FUNCTION_BLOCK EM_DockingInterface EXTENDS EM_Base IMPLEMENTS I_EM_DockingInterface
VAR_INPUT
//Inputs
	i_ref_stSettings : REFERENCE TO ST_SettingsDockingInterface;
	
	//--i_bIlckDockingClampsToClose : BOOL := TRUE; //TRUE = Interlocked
	//--i_bIlckDockingClampsToOpen : BOOL := TRUE; //TRUE = Interlocked
	//--i_bIlckUnlockingPinsToLock : BOOL := TRUE; //TRUE = Interlocked
	//--i_bIlckUnlockingPinsToRelease : BOOL := TRUE; //TRUE = Interlocked
	
	// External interlocks (from outside this EM)
	i_fbExtIlckDockingClampsToClose : FB_Interlock;
	i_fbExtIlckDockingClampsToOpen : FB_Interlock;
	i_fbExtIlckUnlockingPinsToLock : FB_Interlock;
	i_fbExtIlckUnlockingPinsToRelease : FB_Interlock;
	
	i_fbExtIlckInnerDoorOpen : FB_Interlock;
	i_fbExtIlckInnerDoorClose : FB_Interlock;
	
	
	
	i_refTB : REFERENCE TO OBJ_Carrier;	//Mogelijk voor uiteindelijke machine, voor de FUMO's is dit nog niet echt relevant
	//??i_refITF_TB : REFERENCE TO I_Carrier;
END_VAR

VAR_OUTPUT
	q_bStaWarning : BOOL;
END_VAR

VAR
//------------------------------------------//
//Control Modules (Devices)
	s_cmDockingClampsUpper : CM_ValveWithDoubleFB; // Off = Open, On = Close
	s_cmDockingClampsLower : CM_ValveWithDoubleFB; // Off = Open, On = Close
	
	s_cmUnlockingPinUpper : CM_ValveWithFB; // Off = Lock, On = Release
	s_cmUnlockingPinLower : CM_ValveWithFB; // Off = Lock, On = Release
	
	s_cmDoorOpener : CM_ValveWithFB; // Off = Close, On = Open
	s_cmDoorShutter : CM_ValveWithFB; // Off = Open, On = Close
	
//Interlocks	
fbIlckHandlerDockingClampsOpen : FB_InterlockHandler;
fbIlckHandlerDockingClampsClose : FB_InterlockHandler;
fbIlckHandlerUnlockingPinsLock : FB_InterlockHandler;
fbIlckHandlerUnlockingPinsRelease : FB_InterlockHandler;
fbIlckHandlerDoorOpenerClose : FB_InterlockHandler;
fbIlckHandlerDoorOpenerOpen : FB_InterlockHandler;
fbIlckHandlerDoorShutterClose : FB_InterlockHandler;
fbIlckHandlerDoorShutterOpen : FB_InterlockHandler;

//--fbInterlockHandlerDockTB : FB_InterlockHandler;
//--fbInterlockHandlerUndockTB : FB_InterlockHandler;
//--fbInterlockHandlerOpenInnerDoor : FB_InterlockHandler;
//--fbInterlockHandlerCloseInnerDoor : FB_InterlockHandler;	


	
//------------------------------------------//

//------------------------------------------//
//Inputs
	s_diStaDoorAlmostClosed : FB_DigInput;
		
//------------------------------------------//
	
//------------------------------------------//
//Outputs
	s_doCmdClampsUpperHighPressure : FB_DigOutput_2;
	s_doCmdClampsLowerHighPressure : FB_DigOutput_2;

//------------------------------------------//

//Requests
	s_bReqDockBox : BOOL := FALSE;
	s_bReqUndockBox : BOOL := FALSE;
	s_bReqOpenInnerDoor : BOOL := FALSE;
	s_bReqCloseInnerDoor : BOOL := FALSE;
	s_bReqDockingClampsUpperHighPressure : BOOL := FALSE; // True = high pressure
	s_bReqDockingClampsLowerHighPressure : BOOL := FALSE; // True = high pressure
	
	s_bOverruleInterlocks : BOOL := FALSE;
	
//Properties
	s_bStaDocked : BOOL := FALSE;
	s_bStaUndocked : BOOL := FALSE;
	
	s_bStaDockingClampsClosed : BOOL := FALSE;
	s_bStaDockingClampsOpened : BOOL := FALSE;
	s_bStaDockingClampsUpperClosed : BOOL := FALSE;
	s_bStaDockingClampsUpperOpened : BOOL := FALSE;
	s_bStaDockingClampsLowerClosed : BOOL := FALSE;
	s_bStaDockingClampsLowerOpened : BOOL := FALSE;
	
	s_bStaLockingPinUpperReleased : BOOL := FALSE;
	s_bStaLockingPinUpperLocked : BOOL := FALSE;
	s_bStaLockingPinLowerReleased : BOOL := FALSE;
	s_bStaLockingPinLowerLocked : BOOL := FALSE;
		
	s_bStaDoorOpenerOpened : BOOL := FALSE;
	s_bStaDoorOpenerClosed : BOOL := FALSE;
	s_bStaDoorOpenerAlmostClosed : BOOL := FALSE;
	
	s_bStaDoorShutterOpened : BOOL := FALSE;
	s_bStaDoorShutterClosed : BOOL := FALSE;
		
	s_bStaBoxAtPreDockingPosition : BOOL := FALSE;
	s_bStaBoxAtDockedPosition : BOOL := FALSE;
	s_bStaDockingPositionFree : BOOL := FALSE;
	
//Interlockes
	//Higher-layer components
	//--s_bIlckDockTB : BOOL := TRUE;
	//--s_bIlckUndockTB : BOOL := TRUE;	
	//--s_bIlckOpenInnerDoor : BOOL := TRUE;
	//--s_bIlckCloseInnerDoor : BOOL := TRUE;
	
	s_bIlckDockingClampsToClose : BOOL;
	s_bIlckDockingClampsToOpen : BOOL;
	s_bIlckUnlockingPinsToLock : BOOL;
	s_bIlckUnlockingPinsToRelease : BOOL;
	s_bIlckDoorOpenerToClose : BOOL;
	s_bIlckDoorOpenerToOpen : BOOL;
	s_bIlckDoorShutterToClose : BOOL;
	s_bIlckDoorShutterToOpen : BOOL;
	
	s_sMessage : STRING;
	
//Sequencers
	s_eSeqDockingInterface : E_SeqDockingInterface;
	s_fbSeqDockingInterfaceControl : FB_SeqControl;	
	
	s_ePreviousStep : E_SeqDockingInterface;
	s_eResumeStep : E_SeqDockingInterface;
	
	s_tonTimer : TON;
	
	s_bTmpDockingDone : BOOL;
	s_bTmpUndockingDone : BOOL;
	s_bTmpOpenInnerDoorDone : BOOL;
	s_bTmpCloseInnerDoorDone : BOOL;
	
//Alarms
	s_fbAlarmHandlerClosingDoorFailed : FB_AlarmHandler;

	s_bErrClosingDoorFailed : BOOL;
	
//Warnings
	s_fbAlarmHandlerNoBoxPresentAtPreDockingPosition : FB_AlarmHandler;
	s_fbAlarmHandlerNoBoxPresentAtDockedPosition : FB_AlarmHandler;

	s_bWrnNoBoxPresentAtPreDockingPosition : BOOL;
	s_bWrnNoBoxPresentAtDockedPosition : BOOL;
	
	s_bStaWarning : BOOL;
	
//------------------------------------------//
//Params
	s_fbParamTimeoutDockingClamps : FB_HmiParamHandler;
	s_fbParamTimeoutUnlockingPins : FB_HmiParamHandler;
	s_fbParamTimeoutDoorOpener : FB_HmiParamHandler;
	s_fbParamTimeoutDoorShutter : FB_HmiParamHandler;
	
	s_fbParamCompressSealDuration : FB_HmiParamHandler;
	s_fbParamDelayCloseDoorShutterReleasingPins : FB_HmiParamHandler;
	s_fbParamDelayReleaseUnlockingPins : FB_HmiParamHandler;
	s_fbParamDelayOpenDoorShutter : FB_HmiParamHandler;
	s_fbParamDelayOpenDoorOpener : FB_HmiParamHandler;
	s_fbParamDelayCloseDoorShutter : FB_HmiParamHandler;
	s_fbParamDelayLockUnlockingPins : FB_HmiParamHandler;
	
	s_fbParamOpenClampsAfterClosingTimeout : FB_HmiParamHandler;
	s_fbParamCloseClampsAfterEachOther : FB_HmiParamHandler;

//--	//Tool settings
//--	s_fbParamToolHardwareNr				: FB_HmiParamHandler;
//--    s_fbParamToolSoftwareVersion		: FB_HmiParamHandler;

//--	s_fbParamName						: FB_HmiParamHandler;
//--	s_fbParamNumber						: FB_HmiParamHandler;
//--	s_fbParamRevision                   : FB_HmiParamHandler;
	
//--	s_fbParamTeslaMeterIp				: FB_HmiParamHandler;
//--	s_fbParamTeslaMeterPort				: FB_HmiParamHandler;
	
//--	//Product settings (Maybe)
//--	s_fbParamTotalStroke				: FB_HmiParamHandler;
//--	s_fbParamStepStroke					: FB_HmiParamHandler;
//--	s_fbParamAveragingNumberTest		: FB_HmiParamHandler;
	
//--	s_fbParamaMaxMagnitudeCriteria		: FB_HmiParamHandler;
	
//--	s_fbParamRefIduBottom				: FB_HmiParamHandler;
//--	s_fbParamRefItm                     : FB_HmiParamHandler;
//--	s_fbParamRefCenterTpmPipe           : FB_HmiParamHandler;
//--	s_fbParamRefCpValve					: FB_HmiParamHandler;
//------------------------------------------//

//------------------------------------------//
//Variables
	s_sTestResult 						: STRING;
	
	//--s_eCurrentTest						: E_TestMode;
//--	s_stCommandsTesla					: ST_SCPI_TeslaCommands;
	
	
	// Interlocks
	s_bIlckSpeedDoorOuterToOpen 		: BOOL := TRUE;
	s_bIlckSpeedDoorOuterToClose 		: BOOL := TRUE;
	
	s_bIlckDoorLockCleanroomToOpen 		: BOOL := TRUE;
	
//------------------------------------------//

//------------------------------------------//
//Sensor data	
//--	s_aMagneticX						: ARRAY[0..c_nResultDataSize] OF LREAL;
//--	s_aMagneticY						: ARRAY[0..c_nResultDataSize] OF LREAL;
//--	s_aMagneticZ						: ARRAY[0..c_nResultDataSize] OF LREAL;
//--	s_aMagneticMagnitude				: ARRAY[0..c_nResultDataSize] OF LREAL;
//--	s_aProbePositionZ					: ARRAY[0..c_nResultDataSize] OF LREAL;
	
//--	s_sXMLData							: STRING(Param_Project.n_MaxLenghtXmlDbRow*Param_Project.n_NumberofRowsXmlDb);
	
//--	s_aHmi_MagneticTest					: ARRAY[1..3,0..c_nResultDataSize] OF ST_POINT;
	
//	s_aHmi_ProbePositionZ				: ARRAY[1..1,1..GVL_Datalogging.c_nHmiLogSize] OF ST_POINT;
//------------------------------------------//

//------------------------------------------//
//Alarms

//------------------------------------------//

//------------------------------------------//
//Hmi
	s_nToHmiStepNr					: INT;
	s_nToHmiMaxStepNr				: INT;
	s_sToHmiInstructionText			: T_MAXSTRING;
	s_sToHmiProcedure				: T_MAXSTRING;
	
	//Buttons
	s_fbHmiBtnReset					: FB_HmiBtn;
	
	s_fbHmiBtnManualClampsUpperHighPressure : FB_HmiBtn;
	s_fbHmiBtnManualClampsUpperOpen	: FB_HmiBtn;
	s_fbHmiBtnManualClampsUpperClose: FB_HmiBtn;
	
	s_fbHmiBtnManualClampsLowerHighPressure : FB_HmiBtn;
	s_fbHmiBtnManualClampsLowerOpen	: FB_HmiBtn;
	s_fbHmiBtnManualClampsLowerClose: FB_HmiBtn;
	
	s_fbHmiBtnManualPinUpperLock	: FB_HmiBtn;
	s_fbHmiBtnManualPinUpperRelease: FB_HmiBtn;
	
	s_fbHmiBtnManualPinLowerLock	: FB_HmiBtn;
	s_fbHmiBtnManualPinLowerRelease: FB_HmiBtn;
	
	s_fbHmiBtnManualOpenerOpen		: FB_HmiBtn;
	s_fbHmiBtnManualOpenerClose		: FB_HmiBtn;
	
	s_fbHmiBtnManualShutterOpen		: FB_HmiBtn;
	s_fbHmiBtnManualShutterClose	: FB_HmiBtn;
	
	//Buttons for semi-automai
	s_fbHmiBtnDockTB				: FB_HmiBtn;
	s_fbHmiBtnUndockTB				: FB_HmiBtn;
	s_fbHmiBtnOpenInnerDoor			: FB_HmiBtn;
	s_fbHmiBtnCloseInnerDoor		: FB_HmiBtn;
	
	//--s_fbHmiBtnReleaseInnerDoor		: FB_HmiBtn;
	//--s_fbHmiBtnLockInnerDoor			: FB_HmiBtn;
	
	//old
	//--s_fbHmiBtnDock					: FB_HmiBtn;
	//--s_fbHmiBtnUndock				: FB_HmiBtn;
	
	
	//Leds
	s_fbHmiLedClampsUpperPressureSelect : FB_HmiLed;
	s_fbHmiLedClampsLowerPressureSelect : FB_HmiLed;
	
	s_fbHmiLedClampsOpened			: FB_HmiLed;
	s_fbHmiLedClampsClosed			: FB_HmiLed;
	
	s_fbHmiLedPinsLocked			: FB_HmiLed;
	s_fbHmiLedPinsReleased			: FB_HmiLed;
	
	//==
	s_fbHmiLedClampsUpperOpened		: FB_HmiLed;
	s_fbHmiLedClampsUpperClosed		: FB_HmiLed;
	s_fbHmiLedClampsLowerOpened		: FB_HmiLed;
	s_fbHmiLedClampsLowerClosed		: FB_HmiLed;
	
	s_fbHmiLedPinUpperReleased		: FB_HmiLed;
	s_fbHmiLedPinUpperLocked		: FB_HmiLed;
	s_fbHmiLedPinLowerReleased		: FB_HmiLed;
	s_fbHmiLedPinLowerLocked		: FB_HmiLed;
	
	s_fbHmiLedOpenerOpened			: FB_HmiLed;
	s_fbHmiLedOpenerClosed			: FB_HmiLed;
	s_fbHmiLedOpenerAlmostClosed	: FB_HmiLed;
	
	s_fbHmiLedShutterOpened			: FB_HmiLed;
	s_fbHmiLedShutterClosed			: FB_HmiLed;
	
//------------------------------------------//
	s_bTestBool : BOOL;
	s_nTestCnt : UINT;
END_VAR


SUPER^();

METHOD PROTECTED _m_Alarms : BOOL

IF NOT SUPER^._m_Alarms() THEN
	RETURN;
END_IF

// Set error bits

// Alarm Handlers
s_fbAlarmHandlerClosingDoorFailed(
	i_bStaActive := s_bErrClosingDoorFailed, 
	i_eAlarmLevel := E_AlarmLevel.Alarm, 
	i_sAlarmText := CONCAT(i_sEmName, ': Closing inner door failed'));

s_fbAlarmHandlerNoBoxPresentAtPreDockingPosition(
	i_bStaActive := s_bWrnNoBoxPresentAtPreDockingPosition, 
	i_eAlarmLevel := E_AlarmLevel.Warning, 
	i_sAlarmText := CONCAT(i_sEmName, ':No box present AT per-docking position'));
	
s_fbAlarmHandlerNoBoxPresentAtDockedPosition(
	i_bStaActive := s_bWrnNoBoxPresentAtDockedPosition, 
	i_eAlarmLevel := E_AlarmLevel.Warning, 
	i_sAlarmText := CONCAT(i_sEmName, ':No box present at docked position'));

// Reset warnings
IF i_bCmdReset THEN
	s_bWrnNoBoxPresentAtPreDockingPosition := FALSE;
	s_bWrnNoBoxPresentAtDockedPosition := FALSE;
	s_bErrClosingDoorFailed := FALSE;
END_IF	
	
s_bStaError := 
	s_cmDockingClampsUpper.p_bStaError
	OR s_cmDockingClampsLower.p_bStaError
	OR s_cmUnlockingPinUpper.p_bStaError
	OR s_cmUnlockingPinLower.p_bStaError
	OR s_cmDoorOpener.p_bStaError
	OR s_cmDoorShutter.p_bStaError
	OR s_fbAlarmHandlerClosingDoorFailed.q_bStaActive;

s_bStaWarning := 
	s_fbAlarmHandlerNoBoxPresentAtPreDockingPosition.q_bStaActive
	OR s_fbAlarmHandlerNoBoxPresentAtDockedPosition.q_bStaActive
	OR s_cmDockingClampsUpper.p_bStaWarning
	OR s_cmDockingClampsLower.p_bStaWarning
	OR s_cmUnlockingPinUpper.p_bStaWarning
	OR s_cmUnlockingPinLower.p_bStaWarning
	OR s_cmDoorOpener.p_bStaWarning
	OR s_cmDoorShutter.p_bStaWarning;	
	
_m_Alarms := TRUE;
END_METHOD

METHOD PRIVATE _m_AutomaticControl : BOOL

s_fbHmiBtnDockTB.p_bStaVisible := TRUE;
//??s_fbHmiBtnDockTB.p_bStaEnabled := TRUE;

s_fbHmiBtnUndockTB.p_bStaVisible := TRUE;
//??s_fbHmiBtnUndockTB.p_bStaEnabled := TRUE;

s_fbHmiBtnOpenInnerDoor.p_bStaVisible := TRUE;
//??s_fbHmiBtnOpenInnerDoor.p_bStaEnabled := TRUE;

s_fbHmiBtnCloseInnerDoor.p_bStaVisible := TRUE;
//??s_fbHmiBtnCloseInnerDoor.p_bStaEnabled := TRUE;

//--IF s_eSeqDockingInterface <> s_ePreviousStep THEN
//--	s_ePreviousStep := s_eSeqDockingInterface;
//--END_IF

IF s_eSeqDockingInterface <> s_ePreviousStep 
	AND s_eSeqDockingInterface <> E_SeqDockingInterface.ERROR THEN
	s_ePreviousStep := s_eSeqDockingInterface;
END_IF

s_fbSeqDockingInterfaceControl(
	i_nSeqStep := s_eSeqDockingInterface, 
	i_sStepName := TO_STRING(s_eSeqDockingInterface), 
	i_bCmdReset := i_bCmdReset 
					AND (s_eSeqDockingInterface = E_SeqDockingInterface.ERROR) // Only reset/resume sequencer from ERROR state
					AND i_bReqEnable,   
	i_bStaError := s_bStaError OR NOT(i_bReqEnable));
	
s_tonTimer(PT := T#3600S);
	
CASE s_eSeqDockingInterface OF
	
	E_SeqTransport.IDLE:
		s_eSeqDockingInterface := E_SeqDockingInterface.START;
		s_eResumeStep := E_SeqDockingInterface.OPEN_ALL_DOCKING_CLAMPS;
		
	E_SeqDockingInterface.START:
		s_tonTimer.IN := FALSE;
		
		IF _m_SeqStartup() AND s_fbSeqDockingInterfaceControl.q_tmStepTime > T#1S THEN
			s_eSeqDockingInterface := s_eResumeStep;
		END_IF
		
	E_SeqDockingInterface.OPEN_ALL_DOCKING_CLAMPS:
		IF s_fbSeqDockingInterfaceControl.q_bStaEntry THEN	
			s_doCmdClampsUpperHighPressure.i_bStaOutput := FALSE;
			s_doCmdClampsLowerHighPressure.i_bStaOutput := FALSE;
		END_IF
			
		IF s_cmDockingClampsUpper.m_Off() AND s_cmDockingClampsLower.m_Off() THEN
			s_eSeqDockingInterface := E_SeqDockingInterface.READY;
		END_IF
		
	E_SeqDockingInterface.READY:
		IF s_fbSeqDockingInterfaceControl.q_bStaEntry THEN
			//--i_refTB.p_bDockingDone := FALSE;
			i_refTB.p_bUndockingDone S= s_bTmpUndockingDone;
			s_bTmpUndockingDone := FALSE;
		END_IF
	
		IF s_fbHmiBtnDockTB.p_osrBtnPress OR s_bReqDockBox THEN
			IF _m_CmdDockTB(i_refReason := s_sMessage) THEN	
				IF NOT(i_ref_stSettings.bCloseClampsAfterEachOther) THEN 
					s_eSeqDockingInterface := E_SeqDockingInterface.CLOSE_ALL_DOCKING_CLAMPS;
				ELSE
					s_eSeqDockingInterface := E_SeqDockingInterface.CLOSE_LOWER_DOCKING_CLAMPS;
				END_IF
			END_IF
			
			s_bReqDockBox := FALSE;
		END_IF
		
	E_SeqDockingInterface.CLOSE_ALL_DOCKING_CLAMPS:
		IF s_fbSeqDockingInterfaceControl.q_bStaEntry THEN	
			s_doCmdClampsUpperHighPressure.i_bStaOutput := FALSE;
			s_doCmdClampsLowerHighPressure.i_bStaOutput := FALSE;
		END_IF
		
		IF s_cmDockingClampsUpper.m_On() AND s_cmDockingClampsLower.m_On() THEN
			s_eSeqDockingInterface := E_SeqDockingInterface.COMPRESS_ALL_SEAL;
		//ELSE
		//  In case of error all docking clamps will be openeed (this is implemented in error-step)		
		END_IF
	
	E_SeqDockingInterface.COMPRESS_ALL_SEAL:
		IF s_fbSeqDockingInterfaceControl.q_bStaEntry THEN	
			s_doCmdClampsUpperHighPressure.i_bStaOutput := TRUE;
			s_doCmdClampsLowerHighPressure.i_bStaOutput := TRUE;
		END_IF
		
		IF s_fbSeqDockingInterfaceControl.q_tmStepTime >= i_ref_stSettings.tCompressSealDuration THEN
			i_refTB.p_bDockingDone := TRUE;	
			s_eSeqDockingInterface := E_SeqDockingInterface.TB_DOCKED;
		END_IF
	
	E_SeqDockingInterface.CLOSE_LOWER_DOCKING_CLAMPS:
		IF s_fbSeqDockingInterfaceControl.q_bStaEntry THEN	
			s_doCmdClampsLowerHighPressure.i_bStaOutput := FALSE;
		END_IF
		
		IF s_cmDockingClampsLower.m_On() THEN
			s_eSeqDockingInterface := E_SeqDockingInterface.COMPRESS_LOWER_SEAL;
		//ELSE
		//  In case of error all docking clamps will be openeed (this is implemented in error-step)		
		END_IF
	
	E_SeqDockingInterface.COMPRESS_LOWER_SEAL:
		IF s_fbSeqDockingInterfaceControl.q_bStaEntry THEN	
			s_doCmdClampsLowerHighPressure.i_bStaOutput := TRUE;
		END_IF
		
		IF s_fbSeqDockingInterfaceControl.q_tmStepTime >= i_ref_stSettings.tCompressSealDuration THEN
			s_eSeqDockingInterface := E_SeqDockingInterface.CLOSE_UPPER_DOCKING_CLAMPS;
		END_IF
		
	E_SeqDockingInterface.CLOSE_UPPER_DOCKING_CLAMPS:
		IF s_fbSeqDockingInterfaceControl.q_bStaEntry THEN	
			s_doCmdClampsUpperHighPressure.i_bStaOutput := FALSE;
		END_IF
		
		IF s_cmDockingClampsUpper.m_On() THEN
			s_eSeqDockingInterface := E_SeqDockingInterface.COMPRESS_UPPER_SEAL;
		//ELSE
		//  In case of error all docking clamps will be openeed (this is implemented in error-step)		
		END_IF
	
	E_SeqDockingInterface.COMPRESS_UPPER_SEAL:
		IF s_fbSeqDockingInterfaceControl.q_bStaEntry THEN	
			s_doCmdClampsUpperHighPressure.i_bStaOutput := TRUE;
		END_IF
		
		IF s_fbSeqDockingInterfaceControl.q_tmStepTime >= i_ref_stSettings.tCompressSealDuration THEN
			i_refTB.p_bDockingDone := TRUE;	
			s_eSeqDockingInterface := E_SeqDockingInterface.TB_DOCKED;
		END_IF
	
	E_SeqDockingInterface.TB_DOCKED:
		//--IF s_fbSeqDockingInterfaceControl.q_bStaEntry THEN
			//--i_refTB.p_bDockingDone := TRUE;
			//--i_refTB.p_bUndockingDone := FALSE;
		//--END_IF
	
		IF s_fbHmiBtnOpenInnerDoor.p_osrBtnPress OR s_bReqOpenInnerDoor THEN
			IF _m_CmdOpenInnerDoor(i_refReason := s_sMessage) THEN
				IF s_bStaDoorOpenerClosed AND s_bStaDoorShutterClosed THEN
					s_eSeqDockingInterface := E_SeqDockingInterface.RELEASE_UNLOCKING_PINS;
				ELSE
					s_eSeqDockingInterface := E_SeqDockingInterface.CLOSE_DOOR_OPENER_RELEASING_PINS;
				END_IF
			END_IF			
	
			s_bReqOpenInnerDoor := FALSE;
		END_IF
		
		IF s_fbHmiBtnUndockTB.p_osrBtnPress OR s_bReqUndockBox THEN
			IF _m_CmdUndockTB(i_refReason := s_sMessage) THEN	
				s_bTmpUndockingDone := TRUE;
				s_eSeqDockingInterface := E_SeqDockingInterface.OPEN_ALL_DOCKING_CLAMPS;
			END_IF
				
			s_bReqUndockBox := FALSE;	
		END_IF
		
	E_SeqDockingInterface.CLOSE_DOOR_OPENER_RELEASING_PINS:
		s_tonTimer.IN := s_cmDoorOpener.m_Off();
	
		IF s_tonTimer.ET > i_ref_stSettings.tDelayCloseDoorShutterReleasingPins 
			AND s_bStaDoorOpenerAlmostClosed THEN
			s_tonTimer.IN := FALSE;
			s_eSeqDockingInterface := E_SeqDockingInterface.CLOSE_DOOR_SHUTTER_RELEASING_PINS;
		ELSIF s_fbSeqDockingInterfaceControl.q_tmStepTime >= T#10S THEN
			s_bErrClosingDoorFailed := TRUE;
			s_eSeqDockingInterface := E_SeqDockingInterface.ERROR;
		END_IF
		
	E_SeqDockingInterface.CLOSE_DOOR_SHUTTER_RELEASING_PINS:
		//--s_tonTimer.IN := s_cmDoorShutter.m_Off();
		s_tonTimer.IN := s_cmDoorShutter.m_On();
	
		IF s_tonTimer.ET > i_ref_stSettings.tDelayReleaseUnlockingPins THEN
			s_tonTimer.IN := FALSE;
			s_eSeqDockingInterface := E_SeqDockingInterface.RELEASE_UNLOCKING_PINS;
		END_IF	
		
	E_SeqDockingInterface.RELEASE_UNLOCKING_PINS:
		s_tonTimer.IN := (s_cmUnlockingPinUpper.m_On() AND s_cmUnlockingPinLower.m_On());
	
		IF s_tonTimer.ET > i_ref_stSettings.tDelayOpenDoorShutter THEN
			s_tonTimer.IN := FALSE;
			s_eSeqDockingInterface := E_SeqDockingInterface.OPEN_DOOR_SHUTTER;
		END_IF
		
	E_SeqDockingInterface.OPEN_DOOR_SHUTTER:
		//--s_tonTimer.IN := s_cmDoorShutter.m_On();
		s_tonTimer.IN := s_cmDoorShutter.m_Off();
		
		IF s_tonTimer.ET > i_ref_stSettings.tDelayOpenDoorOpener THEN
			s_tonTimer.IN := FALSE;
			s_eSeqDockingInterface := E_SeqDockingInterface.OPEN_DOOR_OPENER;
		END_IF
	
	E_SeqDockingInterface.OPEN_DOOR_OPENER:
		IF s_cmDoorOpener.m_On() THEN
			i_refTB.p_bOpenInnerDoorDone := TRUE;
			s_eSeqDockingInterface := E_SeqDockingInterface.INNER_DOOR_OPENED;
		END_IF
	
	E_SeqDockingInterface.INNER_DOOR_OPENED:
		//--IF s_fbSeqDockingInterfaceControl.q_bStaEntry THEN
			//--i_refTB.p_bOpenInnerDoorDone := TRUE;
			//--i_refTB.p_bCloseInnerDoorDone := FALSE;
		//--END_IF
	
		IF _m_CmdCloseInnerDoor(i_refReason := s_sMessage) THEN
			IF s_fbHmiBtnCloseInnerDoor.p_osrBtnPress OR s_bReqCloseInnerDoor THEN
				s_eSeqDockingInterface := E_SeqDockingInterface.CLOSE_DOOR_OPENER;	
			END_IF
		END_IF	
			
		s_bReqCloseInnerDoor := FALSE;
	
	E_SeqDockingInterface.CLOSE_DOOR_OPENER:
		s_tonTimer.IN := s_cmDoorOpener.m_Off();
		
		IF s_tonTimer.ET > i_ref_stSettings.tDelayCloseDoorShutter
			AND s_bStaDoorOpenerAlmostClosed
			THEN
			s_tonTimer.IN := FALSE;
			s_eSeqDockingInterface := E_SeqDockingInterface.CLOSE_DOOR_SHUTTER;
		ELSIF s_fbSeqDockingInterfaceControl.q_tmStepTime >= T#15S THEN
			s_bErrClosingDoorFailed := TRUE;
			s_eSeqDockingInterface := E_SeqDockingInterface.ERROR;
		END_IF
		
	E_SeqDockingInterface.CLOSE_DOOR_SHUTTER:
		//--s_tonTimer.IN := s_cmDoorShutter.m_Off();
		s_tonTimer.IN := s_cmDoorShutter.m_On();
		
		IF s_tonTimer.ET > i_ref_stSettings.tDelayLockUnlockingPins THEN
			s_tonTimer.IN := FALSE;
			s_eSeqDockingInterface := E_SeqDockingInterface.LOCK_UNLOCKING_PINS;
		END_IF
	
	E_SeqDockingInterface.LOCK_UNLOCKING_PINS:
		IF (s_cmUnlockingPinUpper.m_Off() AND s_cmUnlockingPinLower.m_Off()) THEN
			
			//--i_refTB.p_bOpenInnerDoorDone := FALSE;
			i_refTB.p_bCloseInnerDoorDone := TRUE;
			s_eSeqDockingInterface := E_SeqDockingInterface.TB_DOCKED;
		END_IF
		
	E_SeqDockingInterface.ERROR:
		IF s_fbSeqDockingInterfaceControl.q_bStaEntry THEN
			IF s_ePreviousStep > E_SeqDockingInterface.START
				AND s_ePreviousStep < E_SeqDockingInterface.ERROR THEN
				s_eResumeStep := s_ePreviousStep;
			ELSE 
				s_eResumeStep := E_SeqDockingInterface.OPEN_ALL_DOCKING_CLAMPS;
			END_IF
			
			//Stop controlling all valves
			IF i_ref_stSettings.bOpenClampsAfterClosingTimeout AND_THEN
				s_ePreviousStep = E_SeqDockingInterface.CLOSE_ALL_DOCKING_CLAMPS
				AND (s_cmDockingClampsUpper.p_bStaError OR s_cmDockingClampsLower.p_bStaError) 
				THEN
				//Open all docking clamps if closing on low pressure has failed
				s_doCmdClampsUpperHighPressure.i_bStaOutput := FALSE;
				s_doCmdClampsLowerHighPressure.i_bStaOutput := FALSE;
				s_cmDockingClampsUpper.m_Off();
				s_cmDockingClampsLower.m_Off();
			ELSE
				s_cmDockingClampsUpper.m_Stop();
				s_cmDockingClampsLower.m_Stop();
			END_IF
			
			s_cmUnlockingPinUpper.m_Stop();
			s_cmUnlockingPinLower.m_Stop();
			s_cmDoorOpener.m_Stop();
			s_cmDoorShutter.m_Stop(); 
		END_IF

END_CASE	

s_bReqDockBox := 
s_bReqUndockBox := 
s_bReqOpenInnerDoor := 
s_bReqCloseInnerDoor := FALSE;

//--IF s_eSeqDockingInterface <> s_ePreviousStep 
//--	AND s_eSeqDockingInterface <> E_SeqDockingInterface.ERROR THEN
//--	s_ePreviousStep := s_eSeqDockingInterface;
//--END_IF
END_METHOD

METHOD PRIVATE _m_CmdCloseInnerDoor : BOOL
VAR_INPUT
	i_refReason : REFERENCE TO STRING;
END_VAR

IF NOT i_bReqEnable THEN 
	RETURN;
END_IF

IF s_bIlckDoorOpenerToClose THEN
	i_refReason := CONCAT('Cmd To Close Inner Door: Interlocked - ', fbIlckHandlerDoorOpenerClose.p_sReason);
	_m_CmdCloseInnerDoor := FALSE;
ELSE
	i_refReason := '-';
	_m_CmdCloseInnerDoor := TRUE;
END_IF
END_METHOD

METHOD PRIVATE _m_CmdDockTB : BOOL
VAR_INPUT
	i_refReason : REFERENCE TO STRING;
END_VAR

IF NOT i_bReqEnable THEN 
	RETURN;
END_IF

IF s_bIlckDockingClampsToClose THEN
	i_refReason := CONCAT('Cmd To Dock: Interlocked - ', fbIlckHandlerDockingClampsClose.p_sReason);
	_m_CmdDockTB := FALSE;
ELSE
	i_refReason := '-';
	_m_CmdDockTB := TRUE;
END_IF
END_METHOD

METHOD PRIVATE _m_CmdOpenInnerDoor : BOOL
VAR_INPUT
	i_refReason : REFERENCE TO STRING;
END_VAR

IF NOT i_bReqEnable THEN 
	RETURN;
END_IF

IF s_bIlckDoorShutterToOpen THEN
	i_refReason := CONCAT('Cmd To Open Inner Door: Interlocked - ', fbIlckHandlerDoorShutterOpen.p_sReason);
	_m_CmdOpenInnerDoor := FALSE;
ELSE
	i_refReason := '-';
	_m_CmdOpenInnerDoor := TRUE;
END_IF
END_METHOD

METHOD PRIVATE _m_CmdUndockTB : BOOL
VAR_INPUT
	i_refReason : REFERENCE TO STRING;
END_VAR

IF NOT i_bReqEnable THEN 
	RETURN;
END_IF

IF s_bIlckDockingClampsToOpen THEN
	i_refReason := CONCAT('Cmd To UnDock: Interlocked - ', fbIlckHandlerDockingClampsOpen.p_sReason);
	_m_CmdUndockTB := FALSE;
ELSE
	i_refReason := '-';
	_m_CmdUndockTB := TRUE;
END_IF
END_METHOD

METHOD PROTECTED _m_Devices : BOOL

IF NOT SUPER^._m_Devices() THEN
	RETURN;
END_IF

//--s_diStaBoxAtPreDockingPosition();
//--s_diStaBoxAtDockedPosition();

//--s_cmDockingClamps(
//--	i_bReqEnable := i_bReqEnable,
//--	i_eCtrlMode := i_eCtrlMode,
//--	i_bCmdReset := i_bCmdReset);
//--	//--i_sCmName := 'Docking Clamps');
	
s_cmDockingClampsUpper(
	i_bReqEnable := i_bReqEnable,
	i_eCtrlMode := i_eCtrlMode,
	i_bCmdReset := i_bCmdReset,
	i_bIclkOn := s_bIlckDockingClampsToClose AND NOT(s_bOverruleInterlocks), 
	i_bIclkOff := s_bIlckDockingClampsToOpen AND NOT(s_bOverruleInterlocks));
	
s_cmDockingClampsLower(
	i_bReqEnable := i_bReqEnable,
	i_eCtrlMode := i_eCtrlMode,
	i_bCmdReset := i_bCmdReset,
	i_bIclkOn := s_bIlckDockingClampsToClose AND NOT(s_bOverruleInterlocks), 
	i_bIclkOff := s_bIlckDockingClampsToOpen AND NOT(s_bOverruleInterlocks));	
	
//--s_bStaDockingClampsClosed := s_cmDockingClamps.p_bStaIsClosed;
//--s_bStaDockingClampsOpened := s_cmDockingClamps.p_bStaIsOpened;

s_bStaDockingClampsUpperClosed := s_cmDockingClampsUpper.p_bStaIsOn;
s_bStaDockingClampsUpperOpened := s_cmDockingClampsUpper.p_bStaIsOff;
s_bStaDockingClampsLowerClosed := s_cmDockingClampsLower.p_bStaIsOn;
s_bStaDockingClampsLowerOpened := s_cmDockingClampsLower.p_bStaIsOff;

//--s_cmUnlockingPins(
//--	i_bReqEnable := i_bReqEnable,
//--	i_eCtrlMode := i_eCtrlMode,
//--	i_bCmdReset := i_bCmdReset);
//--	//--i_sCmName := 'Unlocking Pins');
	
s_cmUnlockingPinUpper(
	i_bReqEnable := i_bReqEnable,
	i_eCtrlMode := i_eCtrlMode,
	i_bCmdReset := i_bCmdReset,
	i_bIclkOn := s_bIlckUnlockingPinsToRelease AND NOT(s_bOverruleInterlocks), 
	i_bIclkOff := s_bIlckUnlockingPinsToRelease AND NOT(s_bOverruleInterlocks));
	
s_cmUnlockingPinLower(
	i_bReqEnable := i_bReqEnable,
	i_eCtrlMode := i_eCtrlMode,
	i_bCmdReset := i_bCmdReset,
	i_bIclkOn := s_bIlckUnlockingPinsToRelease AND NOT(s_bOverruleInterlocks), 
	i_bIclkOff := s_bIlckUnlockingPinsToRelease AND NOT(s_bOverruleInterlocks));
	
s_bStaLockingPinUpperReleased := s_cmUnlockingPinUpper.p_bStaIsOn;
s_bStaLockingPinUpperLocked := s_cmUnlockingPinUpper.p_bStaIsOff;
s_bStaLockingPinLowerReleased := s_cmUnlockingPinLower.p_bStaIsOn;
s_bStaLockingPinLowerLocked := s_cmUnlockingPinLower.p_bStaIsOff;	
	
s_cmDoorOpener(
	i_bReqEnable := i_bReqEnable,
	i_eCtrlMode := i_eCtrlMode,
	i_bCmdReset := i_bCmdReset,
	i_bIclkOn := s_bIlckDoorOpenerToOpen AND NOT(s_bOverruleInterlocks), 
	i_bIclkOff := s_bIlckDoorOpenerToClose AND NOT(s_bOverruleInterlocks));

s_bStaDoorOpenerOpened := s_cmDoorOpener.p_bStaIsOn;
s_bStaDoorOpenerClosed := s_cmDoorOpener.p_bStaIsOff;

s_cmDoorShutter(
	i_bReqEnable := i_bReqEnable,
	i_eCtrlMode := i_eCtrlMode,
	i_bCmdReset := i_bCmdReset,
	i_bIclkOn := s_bIlckDoorShutterToClose AND NOT(s_bOverruleInterlocks), 
	i_bIclkOff := s_bIlckDoorShutterToOpen AND NOT(s_bOverruleInterlocks));
	
s_bStaDoorShutterOpened := s_cmDoorShutter.p_bStaIsOff;
s_bStaDoorShutterClosed := s_cmDoorShutter.p_bStaIsOn;

_m_Devices := TRUE;
END_METHOD

METHOD PROTECTED _m_Hmi : BOOL

IF NOT SUPER^._m_Hmi() THEN
	RETURN;
END_IF

//Buttons
//--s_fbHmiBtnDock();
//--s_fbHmiBtnUndock();
s_fbHmiBtnReset();

//Buttons
IF i_bReqEnable AND i_eCtrlMode = E_CtrlMode.AUTOMATIC THEN
	s_fbHmiBtnDockTB.p_bStaEnabled :=
		NOT(s_bIlckDockingClampsToClose)
		AND NOT(s_cmDockingClampsUpper.p_bStaError)
		AND NOT(s_cmDockingClampsLower.p_bStaError)
		AND (s_eSeqDockingInterface = E_SeqDockingInterface.READY);		
		//??AND NOT(s_bReqCenteringTB);
	
	s_fbHmiBtnUnDockTB.p_bStaEnabled :=
		NOT(s_bIlckDockingClampsToOpen)
		AND NOT(s_cmDockingClampsUpper.p_bStaError)
		AND NOT(s_cmDockingClampsLower.p_bStaError)
		AND (s_eSeqDockingInterface = E_SeqDockingInterface.TB_DOCKED);
		//??AND NOT(s_bReqCenteringTB);
	
	s_fbHmiBtnOpenInnerDoor.p_bStaEnabled :=
		NOT(s_bIlckUnlockingPinsToRelease)
		AND NOT(s_bIlckDoorShutterToOpen)
		//AND NOT(s_bIlckDoorOpenerToOpen)
		AND NOT(s_cmUnlockingPinUpper.p_bStaError)
		AND NOT(s_cmUnlockingPinLower.p_bStaError)
		AND NOT(s_cmDoorShutter.p_bStaError)
		AND NOT(s_cmDoorOpener.p_bStaError)
		AND (s_eSeqDockingInterface = E_SeqDockingInterface.TB_DOCKED);
		//??AND NOT(s_bReqCenteringTB);
	
	s_fbHmiBtnCloseInnerDoor.p_bStaEnabled :=
		NOT(s_bIlckUnlockingPinsToLock)
		//--AND NOT(s_bIlckDoorShutterToClose)
		AND NOT(s_bIlckDoorOpenerToClose)
		AND NOT(s_cmUnlockingPinUpper.p_bStaError)
		AND NOT(s_cmUnlockingPinLower.p_bStaError)
		AND NOT(s_cmDoorShutter.p_bStaError)
		AND NOT(s_cmDoorOpener.p_bStaError);
		//??AND NOT(s_bReqCenteringTB);
 
ELSE
	s_fbHmiBtnDockTB.p_bStaEnabled := FALSE;
	s_fbHmiBtnUndockTB.p_bStaEnabled := FALSE;
	s_fbHmiBtnOpenInnerDoor.p_bStaEnabled := FALSE;
	s_fbHmiBtnCloseInnerDoor.p_bStaEnabled := FALSE;
END_IF

s_fbHmiBtnDockTB();
s_fbHmiBtnUndockTB();
	
s_fbHmiBtnOpenInnerDoor();
s_fbHmiBtnCloseInnerDoor();

//Manual control	
s_fbHmiBtnManualClampsUpperHighPressure();
s_fbHmiBtnManualClampsUpperOpen();
s_fbHmiBtnManualClampsUpperClose();

s_fbHmiBtnManualClampsLowerHighPressure();
s_fbHmiBtnManualClampsLowerOpen();
s_fbHmiBtnManualClampsLowerClose();
	
s_fbHmiBtnManualPinUpperLock();
s_fbHmiBtnManualPinUpperRelease();
	
s_fbHmiBtnManualPinLowerLock();
s_fbHmiBtnManualPinLowerRelease();
	
s_fbHmiBtnManualOpenerOpen();
s_fbHmiBtnManualOpenerClose();
	
s_fbHmiBtnManualShutterOpen();
s_fbHmiBtnManualShutterClose();

//Leds
s_fbHmiLedClampsUpperOpened(i_bStaLed := s_bStaDockingClampsUpperOpened);
s_fbHmiLedClampsUpperClosed(i_bStaLed := s_bStaDockingClampsUpperClosed);

s_fbHmiLedClampsLowerOpened(i_bStaLed := s_bStaDockingClampsLowerOpened);
s_fbHmiLedClampsLowerClosed(i_bStaLed := s_bStaDockingClampsLowerClosed);

s_fbHmiLedPinUpperReleased(i_bStaLed := s_bStaLockingPinUpperReleased);
s_fbHmiLedPinUpperLocked(i_bStaLed := s_bStaLockingPinUpperLocked);

s_fbHmiLedPinLowerReleased(i_bStaLed := s_bStaLockingPinLowerReleased);
s_fbHmiLedPinLowerLocked(i_bStaLed := s_bStaLockingPinLowerLocked);
	
s_fbHmiLedOpenerOpened(i_bStaLed := s_bStaDoorOpenerOpened);
s_fbHmiLedOpenerClosed(i_bStaLed := s_bStaDoorOpenerClosed);
s_fbHmiLedOpenerAlmostClosed(i_bStaLed := s_bStaDoorOpenerAlmostClosed);
	
s_fbHmiLedShutterOpened(i_bStaLed := s_bStaDoorShutterOpened);
s_fbHmiLedShutterClosed(i_bStaLed := s_bStaDoorShutterClosed);

_m_Hmi := TRUE;
END_METHOD

METHOD PROTECTED _m_Init : BOOL

IF NOT SUPER^._m_Init() THEN
	RETURN;
END_IF

//Control Modules
//--s_cmDockingClamps.i_bReqEnable := FALSE;
//--s_cmDockingClamps.i_eCtrlMode := E_CtrlMode.IDLE;
//--s_cmDockingClamps.i_sCmName := 'Docking Clamps';
//--s_cmDockingClamps.i_stSettings.tClampsOpenTimeout := T#10S;
//--s_cmDockingClamps.i_stSettings.tClampsCloseTimeout := T#10S;
{warning '#TODO: Dot we need to added configuration parameters? Seperate struct or via settings or dedicateed variables'}

s_cmDockingClampsUpper.i_bReqEnable := FALSE;
s_cmDockingClampsUpper.i_eCtrlMode := E_CtrlMode.IDLE;
s_cmDockingClampsUpper.i_sCmName := 'CM Docking Clamps Upper';
s_cmDockingClampsUpper.i_stSettings.tValveOnTimeout := T#10S;
s_cmDockingClampsUpper.i_stSettings.tValveOnTimeout := T#10S;
s_cmDockingClampsUpper.p_bCfgBiStableValve := FALSE;
s_cmDockingClampsUpper.p_bCfgReverseValve := FALSE;
s_cmDockingClampsUpper.p_sCfgOffName := 'Open';
s_cmDockingClampsUpper.p_sCfgOnName := 'Close';
s_cmDockingClampsUpper.p_sCfgFB1Name := 'Left';
s_cmDockingClampsUpper.p_sCfgFB2Name := 'Right';

s_doCmdClampsUpperHighPressure.i_stSettings.bCfgDelay := FALSE;
s_doCmdClampsUpperHighPressure.i_stSettings.tmOutputDelay := T#0S;

s_cmDockingClampsLower.i_bReqEnable := FALSE;
s_cmDockingClampsLower.i_eCtrlMode := E_CtrlMode.IDLE;
s_cmDockingClampsLower.i_sCmName := 'CM Docking Clamps Lower';
s_cmDockingClampsLower.i_stSettings.tValveOnTimeout := T#10S;
s_cmDockingClampsLower.i_stSettings.tValveOnTimeout := T#10S;
s_cmDockingClampsLower.p_bCfgBiStableValve := FALSE;
s_cmDockingClampsLower.p_bCfgReverseValve := FALSE;
s_cmDockingClampsLower.p_sCfgOffName := 'Open';
s_cmDockingClampsLower.p_sCfgOnName := 'Close';
s_cmDockingClampsLower.p_sCfgFB1Name := 'Left';
s_cmDockingClampsLower.p_sCfgFB2Name := 'Right';

s_doCmdClampsLowerHighPressure.i_stSettings.bCfgDelay := FALSE;
s_doCmdClampsLowerHighPressure.i_stSettings.tmOutputDelay := T#0S;
	
//--s_cmUnlockingPins.i_bReqEnable := FALSE;
//--s_cmUnlockingPins.i_eCtrlMode := E_CtrlMode.IDLE;
//--s_cmUnlockingPins.i_sCmName := 'Unlocking Pins';
//--s_cmUnlockingPins.i_stSettings.tPinsLockTimeout := T#10S;
//--s_cmUnlockingPins.i_stSettings.tPinsUnlockTimeout := T#10S;
{warning '#TODO: Dot we need to added configuration parameters? Seperate struct or via settings or dedicateed variables'}

s_cmUnlockingPinUpper.i_bReqEnable := FALSE;
s_cmUnlockingPinUpper.i_eCtrlMode := E_CtrlMode.IDLE;
s_cmUnlockingPinUpper.i_sCmName := 'CM Unlocking Pin Upper';
s_cmUnlockingPinUpper.i_stSettings.tValveOnTimeout := T#10S;
s_cmUnlockingPinUpper.i_stSettings.tValveOffTimeout := T#10S;
s_cmUnlockingPinUpper.p_bCfgBiStableValve := FALSE;
s_cmUnlockingPinUpper.p_bCfgReverseValve := FALSE;
s_cmUnlockingPinUpper.p_sCfgOffName := 'Lock';
s_cmUnlockingPinUpper.p_sCfgOnName := 'Release';

s_cmUnlockingPinLower.i_bReqEnable := FALSE;
s_cmUnlockingPinLower.i_eCtrlMode := E_CtrlMode.IDLE;
s_cmUnlockingPinLower.i_sCmName := 'CM Unlocking Pin Lower';
s_cmUnlockingPinLower.i_stSettings.tValveOnTimeout := T#10S;
s_cmUnlockingPinLower.i_stSettings.tValveOffTimeout := T#10S;
s_cmUnlockingPinLower.p_bCfgBiStableValve := FALSE;
s_cmUnlockingPinLower.p_bCfgReverseValve := FALSE;
s_cmUnlockingPinLower.p_sCfgOffName := 'Lock';
s_cmUnlockingPinLower.p_sCfgOnName := 'Release';

s_cmDoorOpener.i_bReqEnable := FALSE;
s_cmDoorOpener.i_eCtrlMode := E_CtrlMode.IDLE;
s_cmDoorOpener.i_sCmName := 'CM Door Opener';
s_cmDoorOpener.i_stSettings.tValveOnTimeout := T#10S;
s_cmDoorOpener.i_stSettings.tValveOffTimeout := T#10S;
s_cmDoorOpener.p_bCfgBiStableValve := FALSE;
s_cmDoorOpener.p_bCfgReverseValve := FALSE;
s_cmDoorOpener.p_sCfgOffName := 'Close';
s_cmDoorOpener.p_sCfgOnName := 'Open';

s_diStaDoorAlmostClosed.i_stSettings.tmInputDelay := T#0S;

s_cmDoorShutter.i_bReqEnable := FALSE;
s_cmDoorShutter.i_eCtrlMode := E_CtrlMode.IDLE;
s_cmDoorShutter.i_sCmName := 'CM Door Shutter';
s_cmDoorShutter.i_stSettings.tValveOnTimeout := T#10S;
s_cmDoorShutter.i_stSettings.tValveOffTimeout := T#10S;
s_cmDoorShutter.p_bCfgBiStableValve := FALSE;
s_cmDoorShutter.p_bCfgReverseValve := FALSE;
s_cmDoorShutter.p_sCfgOffName := 'Open';
s_cmDoorShutter.p_sCfgOnName := 'Close';
	

//Interlocks
//Docking Clamps
fbIlckHandlerDockingClampsOpen.i_stInterlockList.arr_Interlocks[1].sReason := 'n/a';
fbIlckHandlerDockingClampsClose.i_stInterlockList.arr_Interlocks[1].sReason := 'n/a';

//Unlockig Pins
fbIlckHandlerUnlockingPinsRelease.i_stInterlockList.arr_Interlocks[1].sReason := 'n/a';
fbIlckHandlerUnlockingPinsLock.i_stInterlockList.arr_Interlocks[1].sReason := 'n/a';

//Door Opener
fbIlckHandlerDoorOpenerClose.i_stInterlockList.arr_Interlocks[1].sReason := 'Door Shutter not opened';
fbIlckHandlerDoorOpenerOpen.i_stInterlockList.arr_Interlocks[1].sReason := 'Door Shutter not opened';

//Door Closer
fbIlckHandlerDoorShutterClose.i_stInterlockList.arr_Interlocks[1].sReason := 'Door Opener not (almost)closed';
fbIlckHandlerDoorShutterOpen.i_stInterlockList.arr_Interlocks[1].sReason := 'n/a';


//---------------------------------//	
	
//----------------------------------//	
//Hmi
	s_fbHmiBtnDockTB.p_eButtontype := E_HmiButtonType.PUSHBUTTON;
	s_fbHmiBtnDockTB.p_bStaVisible := FALSE;
	s_fbHmiBtnDockTB.p_bStaEnabled := FALSE;		
	s_fbHmiBtnDockTB.p_sBtnText := 'Dock TB';
	
	s_fbHmiBtnUndockTB.p_eButtontype := E_HmiButtonType.PUSHBUTTON;
	s_fbHmiBtnUndockTB.p_bStaVisible := FALSE;
	s_fbHmiBtnUndockTB.p_bStaEnabled := FALSE;		
	s_fbHmiBtnUndockTB.p_sBtnText := 'Undocking TB';
	
	s_fbHmiBtnOpenInnerDoor.p_eButtontype := E_HmiButtonType.PUSHBUTTON;
	s_fbHmiBtnOpenInnerDoor.p_bStaVisible := FALSE;
	s_fbHmiBtnOpenInnerDoor.p_bStaEnabled := FALSE;		
	s_fbHmiBtnOpenInnerDoor.p_sBtnText := 'Open Inner Door';
	
	s_fbHmiBtnCloseInnerDoor.p_eButtontype := E_HmiButtonType.PUSHBUTTON;
	s_fbHmiBtnCloseInnerDoor.p_bStaVisible := FALSE;
	s_fbHmiBtnCloseInnerDoor.p_bStaEnabled := FALSE;		
	s_fbHmiBtnCloseInnerDoor.p_sBtnText := 'Close Inner Door';
	
	s_fbHmiBtnReset.p_eButtontype := E_HmiButtonType.PUSHBUTTON;
	s_fbHmiBtnReset.p_bStaVisible := FALSE;
	s_fbHmiBtnReset.p_bStaEnabled := FALSE;		
	s_fbHmiBtnReset.p_sBtnText := 'Reset';
	
	//Manual
	s_fbHmiBtnManualClampsUpperHighPressure.p_eButtontype := E_HmiButtonType.TOGGLEBUTTON;
	s_fbHmiBtnManualClampsUpperHighPressure.p_bStaVisible := FALSE;
	s_fbHmiBtnManualClampsUpperHighPressure.p_bStaEnabled := FALSE;		
	s_fbHmiBtnManualClampsUpperHighPressure.p_sBtnText := 'Pressure Select Upper Clamps';
	
	s_fbHmiBtnManualClampsUpperOpen.p_eButtontype := E_HmiButtonType.PUSHBUTTON;
	s_fbHmiBtnManualClampsUpperOpen.p_bStaVisible := FALSE;
	s_fbHmiBtnManualClampsUpperOpen.p_bStaEnabled := FALSE;		
	s_fbHmiBtnManualClampsUpperOpen.p_sBtnText := 'Open Upper Clamps';
	
	s_fbHmiBtnManualClampsUpperClose.p_eButtontype := E_HmiButtonType.PUSHBUTTON;
	s_fbHmiBtnManualClampsUpperClose.p_bStaVisible := FALSE;
	s_fbHmiBtnManualClampsUpperClose.p_bStaEnabled := FALSE;		
	s_fbHmiBtnManualClampsUpperClose.p_sBtnText := 'Close Upper Clamps';
	
	s_fbHmiBtnManualClampsLowerHighPressure.p_eButtontype := E_HmiButtonType.TOGGLEBUTTON;
	s_fbHmiBtnManualClampsLowerHighPressure.p_bStaVisible := FALSE;
	s_fbHmiBtnManualClampsLowerHighPressure.p_bStaEnabled := FALSE;		
	s_fbHmiBtnManualClampsLowerHighPressure.p_sBtnText := 'Pressure Select Lower Clamps';
	
	s_fbHmiBtnManualClampsLowerOpen.p_eButtontype := E_HmiButtonType.PUSHBUTTON;
	s_fbHmiBtnManualClampsLowerOpen.p_bStaVisible := FALSE;
	s_fbHmiBtnManualClampsLowerOpen.p_bStaEnabled := FALSE;		
	s_fbHmiBtnManualClampsLowerOpen.p_sBtnText := 'Open Lower Clamps';
	
	s_fbHmiBtnManualClampsLowerClose.p_eButtontype := E_HmiButtonType.PUSHBUTTON;
	s_fbHmiBtnManualClampsLowerClose.p_bStaVisible := FALSE;
	s_fbHmiBtnManualClampsLowerClose.p_bStaEnabled := FALSE;		
	s_fbHmiBtnManualClampsLowerClose.p_sBtnText := 'Close Lower Clamps';
	
	s_fbHmiBtnManualPinUpperLock.p_eButtontype := E_HmiButtonType.PUSHBUTTON;
	s_fbHmiBtnManualPinUpperLock.p_bStaVisible := FALSE;
	s_fbHmiBtnManualPinUpperLock.p_bStaEnabled := FALSE;		
	s_fbHmiBtnManualPinUpperLock.p_sBtnText := 'Lock Upper Pins';
	
	s_fbHmiBtnManualPinUpperRelease.p_eButtontype := E_HmiButtonType.PUSHBUTTON;
	s_fbHmiBtnManualPinUpperRelease.p_bStaVisible := FALSE;
	s_fbHmiBtnManualPinUpperRelease.p_bStaEnabled := FALSE;		
	s_fbHmiBtnManualPinUpperRelease.p_sBtnText := 'Release Upper Pins';
	
	s_fbHmiBtnManualPinLowerLock.p_eButtontype := E_HmiButtonType.PUSHBUTTON;
	s_fbHmiBtnManualPinLowerLock.p_bStaVisible := FALSE;
	s_fbHmiBtnManualPinLowerLock.p_bStaEnabled := FALSE;		
	s_fbHmiBtnManualPinLowerLock.p_sBtnText := 'Lock Lower Pins';
	
	s_fbHmiBtnManualPinLowerRelease.p_eButtontype := E_HmiButtonType.PUSHBUTTON;
	s_fbHmiBtnManualPinLowerRelease.p_bStaVisible := FALSE;
	s_fbHmiBtnManualPinLowerRelease.p_bStaEnabled := FALSE;		
	s_fbHmiBtnManualPinLowerRelease.p_sBtnText := 'Release Lower Pins';
	
	s_fbHmiBtnManualOpenerOpen.p_eButtontype := E_HmiButtonType.PUSHBUTTON;
	s_fbHmiBtnManualOpenerOpen.p_bStaVisible := FALSE;
	s_fbHmiBtnManualOpenerOpen.p_bStaEnabled := FALSE;		
	s_fbHmiBtnManualOpenerOpen.p_sBtnText := 'Opener Open';
	
	s_fbHmiBtnManualOpenerClose.p_eButtontype := E_HmiButtonType.PUSHBUTTON;
	s_fbHmiBtnManualOpenerClose.p_bStaVisible := FALSE;
	s_fbHmiBtnManualOpenerClose.p_bStaEnabled := FALSE;		
	s_fbHmiBtnManualOpenerClose.p_sBtnText := 'Opener Close';
	
	s_fbHmiBtnManualShutterOpen.p_eButtontype := E_HmiButtonType.PUSHBUTTON;
	s_fbHmiBtnManualShutterOpen.p_bStaVisible := FALSE;
	s_fbHmiBtnManualShutterOpen.p_bStaEnabled := FALSE;		
	s_fbHmiBtnManualShutterOpen.p_sBtnText := 'Shutter Open';
	
	s_fbHmiBtnManualShutterClose.p_eButtontype := E_HmiButtonType.PUSHBUTTON;
	s_fbHmiBtnManualShutterClose.p_bStaVisible := FALSE;
	s_fbHmiBtnManualShutterClose.p_bStaEnabled := FALSE;		
	s_fbHmiBtnManualShutterClose.p_sBtnText := 'Shutter Close';
	
	//Leds
	s_fbHmiLedClampsUpperPressureSelect.p_bStaVisible := FALSE;
	s_fbHmiLedClampsUpperPressureSelect.p_sToHmiDescriptionLed := 'Pressure Select Upper Clamps';
	
	s_fbHmiLedClampsLowerPressureSelect.p_bStaVisible := FALSE;
	s_fbHmiLedClampsLowerPressureSelect.p_sToHmiDescriptionLed := 'Pressure Select Lower Clamps';
	
	s_fbHmiLedClampsOpened.p_bStaVisible := FALSE;
	s_fbHmiLedClampsOpened.p_sToHmiDescriptionLed := 'Clamps Opened';
		
	s_fbHmiLedClampsClosed.p_bStaVisible := FALSE;
	s_fbHmiLedClampsClosed.p_sToHmiDescriptionLed := 'Clamps Closed';

	//==
	s_fbHmiLedClampsUpperOpened.p_bStaVisible := FALSE;
	s_fbHmiLedClampsUpperOpened.p_sToHmiDescriptionLed := 'Clamps Upper Left Opened';
	
	s_fbHmiLedClampsUpperClosed.p_bStaVisible := FALSE;
	s_fbHmiLedClampsUpperClosed.p_sToHmiDescriptionLed := 'Clamps Upper Left Closed';

	s_fbHmiLedClampsLowerOpened.p_bStaVisible := FALSE;
	s_fbHmiLedClampsLowerOpened.p_sToHmiDescriptionLed := 'Clamps Lower Left Opened';
	
	s_fbHmiLedClampsLowerClosed.p_bStaVisible := FALSE;
	s_fbHmiLedClampsLowerClosed.p_sToHmiDescriptionLed := 'Clamps Lower Left Closed';
	
	
	s_fbHmiLedPinsLocked.p_bStaVisible := FALSE;
	s_fbHmiLedPinsLocked.p_sToHmiDescriptionLed := 'Pins Locked';
	
	s_fbHmiLedPinsReleased.p_bStaVisible := FALSE;
	s_fbHmiLedPinsReleased.p_sToHmiDescriptionLed := 'Pins Unlocked';
	
	//==	
	s_fbHmiLedPinUpperReleased.p_bStaVisible := FALSE;
	s_fbHmiLedPinUpperReleased.p_sToHmiDescriptionLed := 'Unlocking Pin Upper Released';
	s_fbHmiLedPinUpperLocked.p_bStaVisible := FALSE;
	s_fbHmiLedPinUpperLocked.p_sToHmiDescriptionLed := 'Unlocking Pin Upper Locked';
	
	s_fbHmiLedPinLowerReleased.p_bStaVisible := FALSE;
	s_fbHmiLedPinLowerReleased.p_sToHmiDescriptionLed := 'Unlocking Pin Lower Released';
	s_fbHmiLedPinLowerLocked.p_bStaVisible := FALSE;
	s_fbHmiLedPinLowerLocked.p_sToHmiDescriptionLed := 'Unlocking Pin Lower Locked';
	
	s_fbHmiLedOpenerOpened.p_bStaVisible := FALSE;
	s_fbHmiLedOpenerOpened.p_sToHmiDescriptionLed := 'Door Opener Opened';
	s_fbHmiLedOpenerClosed.p_bStaVisible := FALSE;
	s_fbHmiLedOpenerClosed.p_sToHmiDescriptionLed := 'Door Opener Closed';
	s_fbHmiLedOpenerAlmostClosed.p_bStaVisible := FALSE;
	s_fbHmiLedOpenerAlmostClosed.p_sToHmiDescriptionLed := 'Door Opener Almost Closed';
	
	s_fbHmiLedShutterOpened.p_bStaVisible := FALSE;
	s_fbHmiLedShutterOpened.p_sToHmiDescriptionLed := 'Door Shutter Opened';
	s_fbHmiLedShutterClosed.p_bStaVisible := FALSE;
	s_fbHmiLedShutterClosed.p_sToHmiDescriptionLed := 'Door Shutter Closed';
	
//----------------------------------//	
//Initialize all moving averages

//----------------------------------//	

//----------------------------------//	

//Inputs
//--s_diStaBoxAtPreDockingPosition.i_stSettings.tmInputDelay := T#3S;
//--s_diStaBoxAtDockedPosition.i_stSettings.tmInputDelay := T#3S;
//----------------------------------//	

//----------------------------------//	
//Outputs
//--s_doRelayTableDown.i_stSettings.bCfgDelay		:= FALSE;	
//--s_doRelayTableDown.i_stSettings.tmOutputDelay	:= T#0S;	
//----------------------------------//	

_m_Init := TRUE;
END_METHOD

METHOD PROTECTED _m_Inputs : BOOL
IF NOT SUPER^._m_Inputs() THEN
	RETURN;
END_IF

{warning 'TODO# de teksten van onderstaande code mogelijk verplaatsten naar de init method om processor beloasting the verkleinen'}

//Interlocks
//Docking Clamps
fbIlckHandlerDockingClampsOpen.i_stInterlockList.arr_Interlocks[0].bState := i_fbExtIlckDockingClampsToOpen.p_bInterlocked;
fbIlckHandlerDockingClampsOpen.i_stInterlockList.arr_Interlocks[0].sReason := i_fbExtIlckDockingClampsToOpen.p_sReason;
fbIlckHandlerDockingClampsOpen.i_stInterlockList.arr_Interlocks[1].bState := FALSE;
fbIlckHandlerDockingClampsOpen();

fbIlckHandlerDockingClampsClose.i_stInterlockList.arr_Interlocks[0].bState := i_fbExtIlckDockingClampsToClose.p_bInterlocked;
fbIlckHandlerDockingClampsClose.i_stInterlockList.arr_Interlocks[0].sReason := i_fbExtIlckDockingClampsToClose.p_sReason;
fbIlckHandlerDockingClampsClose.i_stInterlockList.arr_Interlocks[1].bState := FALSE;
fbIlckHandlerDockingClampsClose();

//Unlocking Pins
fbIlckHandlerUnlockingPinsLock.i_stInterlockList.arr_Interlocks[0].bState := i_fbExtIlckInnerDoorClose.p_bInterlocked;
fbIlckHandlerUnlockingPinsLock.i_stInterlockList.arr_Interlocks[0].sReason := i_fbExtIlckInnerDoorClose.p_sReason;
fbIlckHandlerUnlockingPinsLock.i_stInterlockList.arr_Interlocks[1].bState := FALSE;
fbIlckHandlerUnlockingPinsLock();

fbIlckHandlerUnlockingPinsRelease.i_stInterlockList.arr_Interlocks[0].bState := i_fbExtIlckInnerDoorOpen.p_bInterlocked;
fbIlckHandlerUnlockingPinsRelease.i_stInterlockList.arr_Interlocks[0].sReason := i_fbExtIlckInnerDoorOpen.p_sReason;
fbIlckHandlerUnlockingPinsRelease.i_stInterlockList.arr_Interlocks[1].bState := FALSE;
fbIlckHandlerUnlockingPinsRelease();

//Door Opener
fbIlckHandlerDoorOpenerClose.i_stInterlockList.arr_Interlocks[0].bState := i_fbExtIlckInnerDoorClose.p_bInterlocked;
fbIlckHandlerDoorOpenerClose.i_stInterlockList.arr_Interlocks[0].sReason := i_fbExtIlckInnerDoorClose.p_sReason;
fbIlckHandlerDoorOpenerClose.i_stInterlockList.arr_Interlocks[1].bState := NOT(s_bStaDoorShutterOpened);
fbIlckHandlerDoorOpenerClose();

fbIlckHandlerDoorOpenerOpen.i_stInterlockList.arr_Interlocks[0].bState := i_fbExtIlckInnerDoorOpen.p_bInterlocked;
fbIlckHandlerDoorOpenerOpen.i_stInterlockList.arr_Interlocks[0].sReason := i_fbExtIlckInnerDoorOpen.p_sReason;
fbIlckHandlerDoorOpenerOpen.i_stInterlockList.arr_Interlocks[1].bState := NOT(s_bStaDoorShutterOpened);

fbIlckHandlerDoorOpenerOpen();

//Door Shutter
fbIlckHandlerDoorShutterClose.i_stInterlockList.arr_Interlocks[0].bState := i_fbExtIlckInnerDoorClose.p_bInterlocked;
fbIlckHandlerDoorShutterClose.i_stInterlockList.arr_Interlocks[0].sReason := i_fbExtIlckInnerDoorClose.p_sReason;
fbIlckHandlerDoorShutterClose.i_stInterlockList.arr_Interlocks[1].bState := NOT(s_bStaDoorOpenerClosed) AND NOT(s_bStaDoorOpenerAlmostClosed); 
fbIlckHandlerDoorShutterClose();

fbIlckHandlerDoorShutterOpen.i_stInterlockList.arr_Interlocks[0].bState := i_fbExtIlckInnerDoorOpen.p_bInterlocked;
fbIlckHandlerDoorShutterOpen.i_stInterlockList.arr_Interlocks[0].sReason := i_fbExtIlckInnerDoorOpen.p_sReason;
fbIlckHandlerDoorShutterClose.i_stInterlockList.arr_Interlocks[1].bState := FALSE;
fbIlckHandlerDoorShutterOpen();

s_bIlckDockingClampsToClose := fbIlckHandlerDockingClampsClose.p_bInterlocked;
s_bIlckDockingClampsToOpen := fbIlckHandlerDockingClampsOpen.p_bInterlocked;
s_bIlckUnlockingPinsToLock := fbIlckHandlerUnlockingPinsLock.p_bInterlocked;
s_bIlckUnlockingPinsToRelease := fbIlckHandlerUnlockingPinsRelease.p_bInterlocked;
s_bIlckDoorOpenerToClose := fbIlckHandlerDoorOpenerClose.p_bInterlocked; //NOT(s_bStaDoorShutterOpened);
s_bIlckDoorOpenerToOpen := fbIlckHandlerDoorOpenerOpen.p_bInterlocked; //NOT(s_bStaDoorShutterOpened);
s_bIlckDoorShutterToClose := fbIlckHandlerDoorShutterClose.p_bInterlocked; //NOT(s_bStaDoorOpenerClosed) AND NOT(s_bStaDoorOpenerAlmostClosed);
s_bIlckDoorShutterToOpen := fbIlckHandlerDoorShutterOpen.p_bInterlocked; //FALSE;

//--s_bIlckDockTB := fbIlckHandlerDockingClampsClose.p_bInterlocked;
//--s_bIlckUnDockTB := fbIlckHandlerDockingClampsOpen.p_bInterlocked;

//--s_bIlckOpenInnerDoor
//--	:= fbIlckHandlerUnlockingPinsRelease.p_bInterlocked
//--	OR fbIlckHandlerDoorOpenerOpen.p_bInterlocked
//--	OR fbIlckHandlerDoorShutterOpen.p_bInterlocked;
//--s_bIlckCloseInnerDoor
//--	:= fbIlckHandlerUnlockingPinsLock.p_bInterlocked
//--	OR fbIlckHandlerDoorOpenerClose.p_bInterlocked
//--	OR fbIlckHandlerDoorShutterClose.p_bInterlocked;

//Docking Clamps
IF s_bIlckDockingClampsToOpen THEN
	s_cmDockingClampsUpper.p_sInterlockedReasonOff := fbIlckHandlerDockingClampsOpen.p_sReason;
	s_cmDockingClampsLower.p_sInterlockedReasonOff := fbIlckHandlerDockingClampsOpen.p_sReason;
ELSE
	s_cmDockingClampsUpper.p_sInterlockedReasonOff := '-';
	s_cmDockingClampsLower.p_sInterlockedReasonOff := '-';
END_IF

IF s_bIlckDockingClampsToClose THEN
	s_cmDockingClampsUpper.p_sInterlockedReasonOn := fbIlckHandlerDockingClampsClose.p_sReason;
	s_cmDockingClampsLower.p_sInterlockedReasonOn := fbIlckHandlerDockingClampsClose.p_sReason;
ELSE
	s_cmDockingClampsUpper.p_sInterlockedReasonOn := '-';
	s_cmDockingClampsLower.p_sInterlockedReasonOn := '-';
END_IF

//Unlocking Pins
IF s_bIlckUnlockingPinsToLock THEN
	s_cmUnlockingPinUpper.p_sInterlockedReasonOff := fbIlckHandlerUnlockingPinsLock.p_sReason;
	s_cmUnlockingPinLower.p_sInterlockedReasonOff := fbIlckHandlerUnlockingPinsLock.p_sReason;
ELSE
	s_cmUnlockingPinUpper.p_sInterlockedReasonOff := '-';
	s_cmUnlockingPinLower.p_sInterlockedReasonOff := '-';
END_IF

IF s_bIlckUnlockingPinsToRelease THEN
	s_cmUnlockingPinUpper.p_sInterlockedReasonOn := fbIlckHandlerUnlockingPinsRelease.p_sReason;
	s_cmUnlockingPinLower.p_sInterlockedReasonOn := fbIlckHandlerUnlockingPinsRelease.p_sReason;
ELSE
	s_cmUnlockingPinUpper.p_sInterlockedReasonOn := '-';
	s_cmUnlockingPinLower.p_sInterlockedReasonOn := '-';
END_IF

//Door Opener
IF s_bIlckDoorOpenerToClose THEN
	s_cmDoorOpener.p_sInterlockedReasonOff := fbIlckHandlerDoorOpenerClose.p_sReason;
ELSE
	s_cmDoorOpener.p_sInterlockedReasonOff := '-';
END_IF

IF s_bIlckDoorOpenerToOpen THEN
	s_cmDoorOpener.p_sInterlockedReasonOn := fbIlckHandlerDoorOpenerOpen.p_sReason;
ELSE
	s_cmDoorOpener.p_sInterlockedReasonOn := '-';
END_IF

//Door Shutter
IF s_bIlckDoorShutterToClose THEN
	s_cmDoorShutter.p_sInterlockedReasonOff := fbIlckHandlerDoorShutterClose.p_sReason;
ELSE
	s_cmDoorShutter.p_sInterlockedReasonOff := '-';
END_IF

IF s_bIlckDoorShutterToOpen THEN
	s_cmDoorShutter.p_sInterlockedReasonOn := fbIlckHandlerDoorShutterOpen.p_sReason;
ELSE
	s_cmDoorShutter.p_sInterlockedReasonOn := '-';
END_IF


(* --
s_cmDockingClampsUpper.p_sInterlockedReasonOn := 'n/a';
s_cmDockingClampsLower.p_sInterlockedReasonOn := 'n/a';

IF s_bIlckDockTB THEN
	s_cmDockingClampsUpper.p_sInterlockedReasonOn := fbInterlockHandlerDockTB.p_sReason;
	s_cmDockingClampsLower.p_sInterlockedReasonOn := fbInterlockHandlerDockTB.p_sReason;
ELSIF
	s_bIlckUndockTB THEN
	s_cmDockingClampsUpper.p_sInterlockedReasonOn := fbInterlockHandlerUnDockTB.p_sReason;
	s_cmDockingClampsLower.p_sInterlockedReasonOn := fbInterlockHandlerUnDockTB.p_sReason;
ELSE
	s_cmDockingClampsUpper.p_sInterlockedReasonOn := '-';
	s_cmDockingClampsLower.p_sInterlockedReasonOn := '-';
END_IF


s_cmUnlockingPinUpper.p_sInterlockedReasonOn := 'n/a';
s_cmUnlockingPinLower.p_sInterlockedReasonOn := 'n/a';

IF NOT(s_bStaDoorShutterOpened) THEN
	s_cmDoorOpener.p_sInterlockedReasonOn := 'Door shutter not opened';
ELSE
	s_cmDoorOpener.p_sInterlockedReasonOn := '-';
END_IF
	
IF NOT(s_bStaDoorOpenerClosed) AND NOT(s_bStaDoorOpenerAlmostClosed) THEN
	s_cmDoorShutter.p_sInterlockedReasonOn := 'Door opener not (almost) closed';
ELSE	
	s_cmDoorShutter.p_sInterlockedReasonOn := '-';
END_IF
-- *)


//--s_diStaBoxAtPreDockingPosition();
//--s_diStaBoxAtDockedPosition();

//--s_bStaBoxAtPreDockingPosition := s_diStaBoxAtPreDockingPosition.p_bStaInputDelayed AND NOT(s_diStaBoxAtDockedPosition.p_bStaInputDelayed);
//--s_bStaBoxAtDockedPosition := s_diStaBoxAtPreDockingPosition.p_bStaInputDelayed AND s_diStaBoxAtDockedPosition.p_bStaInputDelayed;
//--s_bStaDockingPositionFree := NOT(s_bStaBoxAtPreDockingPosition) AND NOT(s_bStaBoxAtDockedPosition);

s_diStaDoorAlmostClosed();

s_bStaDoorOpenerAlmostClosed := s_diStaDoorAlmostClosed.p_bStaInputDelayed;

_m_Inputs := TRUE;
END_METHOD

METHOD PRIVATE _m_ManualControl : BOOL

// Manual control has been implemented into lower layer control modules
IF s_fbHmiBtnManualClampsUpperHighPressure.p_osrBtnPress THEN
	s_doCmdClampsUpperHighPressure.i_bStaOutput := TRUE;
ELSIF s_fbHmiBtnManualClampsUpperHighPressure.p_osfBtnPress THEN
	s_doCmdClampsUpperHighPressure.i_bStaOutput := FALSE;
END_IF

IF s_fbHmiBtnManualClampsLowerHighPressure.p_osrBtnPress THEN
	s_doCmdClampsLowerHighPressure.i_bStaOutput := TRUE;
ELSIF s_fbHmiBtnManualClampsLowerHighPressure.p_osfBtnPress THEN
	s_doCmdClampsLowerHighPressure.i_bStaOutput := FALSE;
END_IF
END_METHOD

METHOD PROTECTED _m_Outputs : BOOL

IF NOT SUPER^._m_Outputs() THEN
	RETURN;
END_IF

s_doCmdClampsUpperHighPressure(i_eCtrlMode := i_eCtrlMode);
s_doCmdClampsLowerHighPressure(i_eCtrlMode := i_eCtrlMode);

s_bStaDocked	:=	s_cmDockingClampsUpper.p_bStaIsOn AND s_doCmdClampsUpperHighPressure.p_bStaOutput
				AND s_cmDockingClampsLower.p_bStaIsOn AND s_doCmdClampsLowerHighPressure.p_bStaOutput;  
s_bStaUndocked 	:= s_cmDockingClampsUpper.p_bStaIsOff AND s_cmDockingClampsLower.p_bStaIsOff;




q_bStaWarning := s_bStaWarning;

_m_Outputs := TRUE;
END_METHOD

METHOD PROTECTED _m_Params : BOOL

IF NOT SUPER^._m_Params() THEN
	RETURN;
END_IF

//Paramaters
s_fbParamTimeoutDockingClamps(
	i_fDefaultValue := ,
	i_sName := CONCAT(i_sEmName, ': Timeout Docking Clamps'),
	i_nArrayFolderIndex := 1,
	i_bIsNumber := TRUE);
	
s_fbParamTimeoutUnlockingPins(
	i_fDefaultValue := ,
	i_sName := CONCAT(i_sEmName, ': Timeout Unlocking Pins'),
	i_nArrayFolderIndex := 1,
	i_bIsNumber := TRUE);
	
s_fbParamTimeoutDoorOpener(
	i_fDefaultValue := ,
	i_sName := CONCAT(i_sEmName, ': Timeout Door Opener'),
	i_nArrayFolderIndex := 1,
	i_bIsNumber := TRUE);
	
s_fbParamTimeoutDoorShutter(
	i_fDefaultValue := ,
	i_sName := CONCAT(i_sEmName, ': Timeout Door Shutter'),
	i_nArrayFolderIndex := 1,
	i_bIsNumber := TRUE);
	
s_fbParamCompressSealDuration(
	i_fDefaultValue := ,
	i_sName := CONCAT(i_sEmName, ': Compress Seal Duration'),
	i_nArrayFolderIndex := 1,
	i_bIsNumber := TRUE);
	
s_fbParamDelayCloseDoorShutterReleasingPins(
	i_fDefaultValue := ,
	i_sName := CONCAT(i_sEmName, ': Delay Close Door Shutter Releasing Pins'),
	i_nArrayFolderIndex := 1,
	i_bIsNumber := TRUE);
	
s_fbParamDelayReleaseUnlockingPins(
	i_fDefaultValue := ,
	i_sName := CONCAT(i_sEmName, ': Delay Release Unlocking Pins'),
	i_nArrayFolderIndex := 1,
	i_bIsNumber := TRUE);
	
s_fbParamDelayOpenDoorShutter(
	i_fDefaultValue := ,
	i_sName := CONCAT(i_sEmName, ': Delay Open Door Shutter'),
	i_nArrayFolderIndex := 1,
	i_bIsNumber := TRUE);
	
s_fbParamDelayOpenDoorOpener(
	i_fDefaultValue := ,
	i_sName := CONCAT(i_sEmName, ': Delay Open Door Opener'),
	i_nArrayFolderIndex := 1,
	i_bIsNumber := TRUE);
	
s_fbParamDelayCloseDoorShutter(
	i_fDefaultValue := ,
	i_sName := CONCAT(i_sEmName, ': Delay Close Door Shutter'),
	i_nArrayFolderIndex := 1,
	i_bIsNumber := TRUE);
	
s_fbParamDelayLockUnlockingPins(
	i_fDefaultValue := ,
	i_sName := CONCAT(i_sEmName, ': Delay Lock Unlocking Pins'),
	i_nArrayFolderIndex := 1,
	i_bIsNumber := TRUE);
	
s_fbParamOpenClampsAfterClosingTimeout(
	i_fDefaultValue := ,
	i_sName := CONCAT(i_sEmName, ': Open Clamps After Closing Timeout'),
	i_nArrayFolderIndex := 1,
	i_bIsNumber := TRUE);
	
s_fbParamCloseClampsAfterEachOther(
	i_fDefaultValue := ,
	i_sName := CONCAT(i_sEmName, ': Close Clamps After Each Other'),
	i_nArrayFolderIndex := 1,
	i_bIsNumber := TRUE);

//Write to settings	

i_ref_stSettings.tTimeoutDockingClamps := LREAL_TO_TIME(s_fbParamTimeoutDockingClamps.p_fValue);
i_ref_stSettings.tTimeoutUnlockingPins := LREAL_TO_TIME(s_fbParamTimeoutUnlockingPins.p_fValue);
i_ref_stSettings.tTimeoutDoorOpener := LREAL_TO_TIME(s_fbParamTimeoutDoorOpener.p_fValue);
i_ref_stSettings.tTimeoutDoorShutter := LREAL_TO_TIME(s_fbParamTimeoutDoorShutter.p_fValue);
	
i_ref_stSettings.tCompressSealDuration := LREAL_TO_TIME(s_fbParamCompressSealDuration.p_fValue);
i_ref_stSettings.tDelayCloseDoorShutterReleasingPins := LREAL_TO_TIME(s_fbParamDelayCloseDoorShutterReleasingPins.p_fValue);
i_ref_stSettings.tDelayReleaseUnlockingPins := LREAL_TO_TIME(s_fbParamDelayReleaseUnlockingPins.p_fValue);
i_ref_stSettings.tDelayOpenDoorShutter := LREAL_TO_TIME(s_fbParamDelayOpenDoorShutter.p_fValue);
i_ref_stSettings.tDelayOpenDoorOpener := LREAL_TO_TIME(s_fbParamDelayOpenDoorOpener.p_fValue);
i_ref_stSettings.tDelayCloseDoorShutter := LREAL_TO_TIME(s_fbParamDelayCloseDoorShutter.p_fValue);
i_ref_stSettings.tDelayLockUnlockingPins := LREAL_TO_TIME(s_fbParamDelayLockUnlockingPins.p_fValue);
	
i_ref_stSettings.bOpenClampsAfterClosingTimeout := LREAL_TO_BOOL(s_fbParamOpenClampsAfterClosingTimeout.p_fValue);
i_ref_stSettings.bCloseClampsAfterEachOther := LREAL_TO_BOOL(s_fbParamCloseClampsAfterEachOther.p_fValue);
	
_m_Params := TRUE;
END_METHOD

METHOD PRIVATE _m_SeqStartup : BOOL

s_bReqDockingClampsUpperHighPressure := FALSE; //Low pressure 
s_bReqDockingClampsLowerHighPressure := FALSE; //Low pressure

(*
IF s_cmDoorOpener.m_Off() OR s_bStaDoorOpenerAlmostClosed THEN //Close Door Opener
	IF s_cmDoorShutter.m_On()THEN //Close Door Shutter
		IF s_cmUnlockingPinUpper.m_Off() AND s_cmUnlockingPinLower.m_Off() THEN //Lock Unlocking Pins
			IF s_cmDockingClampsUpper.m_Off() AND s_cmDockingClampsLower.m_Off() THEN // Open Docking Clamps
				_m_SeqStartup := TRUE;
			END_IF
		END_IF						
	END_IF
END_IF
*)

IF s_cmDoorOpener.m_Off() OR s_bStaDoorOpenerAlmostClosed THEN //Close Door Opener
	IF s_cmDoorShutter.m_On() THEN //Close Door Shutter
		IF s_cmUnlockingPinUpper.m_Off() AND s_cmUnlockingPinLower.m_Off() THEN //Lock Unlocking Pins
			IF s_cmDockingClampsUpper.m_Off() AND s_cmDockingClampsLower.m_Off() THEN // Open Docking Clamps
				_m_SeqStartup := TRUE;
			END_IF
		END_IF						
	END_IF
END_IF
END_METHOD

METHOD PUBLIC m_Main : BOOL

IF NOT SUPER^.m_Main() THEN
	RETURN;
END_IF

CASE i_eCtrlMode OF

	E_CtrlMode.IDLE:
		//--s_cmDockingClamps.m_Stop();
		//--s_cmUnlockingPins.m_Stop();
		
		s_bReqDockBox := FALSE;
		s_bReqUndockBox := FALSE;
		
	E_CtrlMode.AUTOMATIC:
	
		//Let pressure selection toggle follow automatic state
		IF s_doCmdClampsUpperHighPressure.p_bStaOutput THEN
			s_fbHmiBtnManualClampsUpperHighPressure.m_On();
		ELSE
			s_fbHmiBtnManualClampsUpperHighPressure.m_Off();	
		END_IF
		
		IF s_doCmdClampsLowerHighPressure.p_bStaOutput THEN
			s_fbHmiBtnManualClampsLowerHighPressure.m_On();
		ELSE
			s_fbHmiBtnManualClampsLowerHighPressure.m_Off();	
		END_IF
	
		//Execute automatic control
		_m_AutomaticControl();
	
(*		s_fbSeqDockingInterface(
			i_nSeqStep := s_eSeqDockingInterface, 
			i_sStepName := TO_STRING(s_fbSeqDockingInterface.q_eActState), 
			i_bCmdReset := i_bCmdReset, 
			i_bStaError := s_bStaError);
	
		CASE s_eSeqDockingInterface OF
			
			E_SeqDockingInterface.IDLE:
			
				IF s_bReqDockBox THEN
					//--IF s_diStaBoxAtPreDockingPosition.p_bStaInputDelayed THEN
					IF s_bStaBoxAtPreDockingPosition THEN	
						s_bStaUndockingDone := FALSE;
						s_eSeqDockingInterface := E_SeqDockingInterface.DOCKING_CLOSE_CLAMPS;
					ELSE
						s_bWrnNoBoxPresentAtPreDockingPosition := TRUE;	
					END_IF
				END_IF
				
				IF s_bReqUndockBox THEN
					IF s_diStaBoxAtDockedPosition.p_bStaInputDelayed THEN
						s_bStaDockingDone := FALSE;
						s_eSeqDockingInterface := E_SeqDockingInterface.UNDOCKING_LOCK_DOOR;
					ELSE
						s_bWrnNoBoxPresentAtDockedPosition := TRUE;	
					END_IF	
				END_IF
			
				// Seperatly opening/closing the clamps is nessescary to move these out of the way for moving of the outer door
				// Clamps must be closed before the outer door can be moved
				IF s_bReqClosDockingClamps THEN
					s_eSeqDockingInterface := E_SeqDockingInterface.ONLY_CLOSE_CLAMPS;
				END_IF
				
				IF s_bReqOpenDockingClamps THEN
					s_eSeqDockingInterface := E_SeqDockingInterface.ONLY_OPEN_CLAMPS;
				END_IF
				
			E_SeqDockingInterface.DOCKING_CLOSE_CLAMPS:
				
				IF s_fbSeqDockingInterface.q_bStaEntry THEN 
					s_cmDockingClamps.m_Close();
				END_IF
				
				IF s_cmDockingClamps.p_bStaIsClosed THEN
					s_eSeqDockingInterface := E_SeqDockingInterface.DOCKING_UNLOCK_DOOR;
				ELSIF s_cmDockingClamps.p_bStaError THEN 
					s_eSeqDockingInterface := E_SeqDockingInterface.ERROR;
					// write down some info?
				ELSIF (s_fbSeqDockingInterface.q_tmStepTime >= i_stSettings.tTimeoutDockingClamps) THEN
 					s_eSeqDockingInterface := E_SeqDockingInterface.ERROR;
					// write down some info?
				END_IF
			
			E_SeqDockingInterface.DOCKING_UNLOCK_DOOR:
			
				IF s_fbSeqDockingInterface.q_bStaEntry THEN 
					s_cmUnlockingPins.m_Unlock();
				END_IF
				
				IF s_cmUnlockingPins.p_bStaIsUnlocked THEN
					s_eSeqDockingInterface := E_SeqDockingInterface.DOCKING_DONE;
				ELSIF s_cmUnlockingPins.p_bStaError THEN 
					s_eSeqDockingInterface := E_SeqDockingInterface.ERROR;
					// write down some info?
				ELSIF (s_fbSeqDockingInterface.q_tmStepTime >= i_stSettings.tTimeoutUnlockingPins) THEN
 					s_eSeqDockingInterface := E_SeqDockingInterface.ERROR;
					// write down some info?
				END_IF
			
			E_SeqDockingInterface.DOCKING_DONE:
				s_bStaDockingDone := TRUE;
				s_eSeqDockingInterface := E_SeqDockingInterface.IDLE;
			
			E_SeqDockingInterface.UNDOCKING_LOCK_DOOR:
			
				IF s_fbSeqDockingInterface.q_bStaEntry THEN 
					s_cmUnlockingPins.m_Lock();
				END_IF
				
				IF s_cmUnlockingPins.p_bStaIsLocked THEN
					s_eSeqDockingInterface := E_SeqDockingInterface.UNDOCKING_OPEN_CLAMPS;
				ELSIF s_cmUnlockingPins.p_bStaError THEN 
					s_eSeqDockingInterface := E_SeqDockingInterface.ERROR;
					// write down some info?
				ELSIF (s_fbSeqDockingInterface.q_tmStepTime >= i_stSettings.tTimeoutUnlockingPins) THEN
 					s_eSeqDockingInterface := E_SeqDockingInterface.ERROR;
					// write down some info?
				END_IF
				
			E_SeqDockingInterface.UNDOCKING_OPEN_CLAMPS:
			
				IF s_fbSeqDockingInterface.q_bStaEntry THEN 
					s_cmDockingClamps.m_Open();
				END_IF
				
				IF s_cmDockingClamps.p_bStaIsOpened THEN
					s_eSeqDockingInterface := E_SeqDockingInterface.UNDOCKING_DONE;
				ELSIF s_cmDockingClamps.p_bStaError THEN 
					s_eSeqDockingInterface := E_SeqDockingInterface.ERROR;
					// write down some info?
				ELSIF (s_fbSeqDockingInterface.q_tmStepTime >= i_stSettings.tTimeoutDockingClamps) THEN
 					s_eSeqDockingInterface := E_SeqDockingInterface.ERROR;
					// write down some info?
				END_IF
				
			E_SeqDockingInterface.UNDOCKING_DONE:
				s_bStaUndockingDone := TRUE;
				s_eSeqDockingInterface := E_SeqDockingInterface.IDLE;
				
			E_SeqDockingInterface.ONLY_CLOSE_CLAMPS:
			
				IF s_fbSeqDockingInterface.q_bStaEntry THEN
					s_cmDockingClamps.m_Close();
				END_IF
			
				IF s_cmDockingClamps.p_bStaIsClosed THEN
					s_eSeqDockingInterface := E_SeqDockingInterface.IDLE;
				ELSIF (s_fbSeqDockingInterface.q_tmStepTime >= i_stSettings.tTimeoutDockingClamps) THEN
 					s_eSeqDockingInterface := E_SeqDockingInterface.ERROR;
					// write down some info?
				END_IF
			
			E_SeqDockingInterface.ONLY_OPEN_CLAMPS:	
				
				IF s_fbSeqDockingInterface.q_bStaEntry THEN
					s_cmDockingClamps.m_Open();
				END_IF
			
				IF s_cmDockingClamps.p_bStaIsOpened THEN
					s_eSeqDockingInterface := E_SeqDockingInterface.IDLE;
				ELSIF (s_fbSeqDockingInterface.q_tmStepTime >= i_stSettings.tTimeoutDockingClamps) THEN
 					s_eSeqDockingInterface := E_SeqDockingInterface.ERROR;
					// write down some info?
				END_IF
				
			E_SeqDockingInterface.READY:
				;
			
			E_SeqDockingInterface.ERROR:
				
				IF i_bCmdReset THEN
					//Reset errors (probebly alredy done in the methode devices)
					//--cmValveDockingClampsUpper.i_bCmdReset := TRUE;
				
					s_eSeqDockingInterface := E_SeqDockingInterface.IDLE;
				END_IF
				
		END_CASE		
*)	
		
	E_CtrlMode.MANUAL:
		//Reset automatic sequencer
		s_eSeqDockingInterface := E_SeqDockingInterface.IDLE;
		
		_m_ManualControl();

END_CASE
END_METHOD

{attribute 'TcRpcEnable'}
METHOD PUBLIC m_ReqCloseInnerDoor : BOOL

IF NOT i_bReqEnable THEN 
	RETURN;
END_IF

s_bReqDockBox := FALSE;
s_bReqUndockBox := FALSE;
s_bReqOpenInnerDoor := FALSE;
s_bReqCloseInnerDoor := TRUE;

m_ReqCloseInnerDoor := TRUE;
END_METHOD

{attribute 'TcRpcEnable'}
METHOD PUBLIC m_ReqDockTB : BOOL

IF NOT i_bReqEnable THEN 
	RETURN;
END_IF

s_bReqDockBox := TRUE;
s_bReqUndockBox := FALSE;
s_bReqOpenInnerDoor := FALSE;
s_bReqCloseInnerDoor := FALSE;

m_ReqDockTB := TRUE;
END_METHOD

{attribute 'TcRpcEnable'}
METHOD PUBLIC m_ReqOpenInnerDoor : BOOL

IF NOT i_bReqEnable THEN 
	RETURN;
END_IF

s_bReqDockBox := FALSE;
s_bReqUndockBox := FALSE;
s_bReqOpenInnerDoor := TRUE;
s_bReqCloseInnerDoor := FALSE;

m_ReqOpenInnerDoor := TRUE;
END_METHOD

{attribute 'TcRpcEnable'}
METHOD PUBLIC m_ReqUndockTB : BOOL

IF NOT i_bReqEnable THEN 
	RETURN;
END_IF

s_bReqDockBox := FALSE;
s_bReqUndockBox := TRUE;
s_bReqOpenInnerDoor := FALSE;
s_bReqCloseInnerDoor := FALSE;

m_ReqUndockTB := TRUE;
END_METHOD

PROPERTY PUBLIC p_bStaBoxAtDockedPosition : BOOL
GET

p_bStaBoxAtDockedPosition := s_bStaBoxAtDockedPosition;
END_GET
END_PROPERTY

PROPERTY PUBLIC p_bStaBoxAtPreDockingPosition : BOOL
GET

p_bStaBoxAtPreDockingPosition := s_bStaBoxAtPreDockingPosition;
END_GET
END_PROPERTY

PROPERTY PUBLIC p_bStaDocked : BOOL
GET

p_bStaDocked := s_bStaDocked;
END_GET
END_PROPERTY

PROPERTY PUBLIC p_bStaDockingClampsClosed : BOOL
GET

p_bStaDockingClampsClosed := s_bStaDockingClampsClosed;
END_GET
END_PROPERTY

PROPERTY PUBLIC p_bStaDockingClampsOpened : BOOL
GET

p_bStaDockingClampsOpened := s_bStaDockingClampsOpened;
END_GET
END_PROPERTY

PROPERTY PUBLIC p_bStaDockingPositionFree : BOOL
GET

p_bStaDockingPositionFree := s_bStaDockingPositionFree;
END_GET
END_PROPERTY

PROPERTY PUBLIC p_bStaInnerDoorClosedAndLocked : BOOL
GET

p_bStaInnerDoorClosedAndLocked := 
	s_bStaLockingPinLowerLocked
AND s_bStaLockingPinUpperLocked
AND s_bStaDoorOpenerClosed
AND s_bStaDoorShutterClosed;
END_GET
END_PROPERTY

PROPERTY PUBLIC p_bStaInnerDoorOpenedAndReleased : BOOL
GET

p_bStaInnerDoorOpenedAndReleased := 
	s_bStaLockingPinLowerReleased
AND s_bStaLockingPinUpperReleased
AND s_bStaDoorOpenerOpened
AND s_bStaDoorShutterOpened;
END_GET
END_PROPERTY

PROPERTY PUBLIC p_bStaUndocked : BOOL
GET

p_bStaUndocked := s_bStaUndocked;
END_GET
END_PROPERTY

END_FUNCTION_BLOCK

(* stored: Version 1.1.0.1, ProductVersion 3.1.4024.12
   POU EM_DockingInterface: Id {1a98308c-f0e0-4a53-963d-dfa6a727e4cb}, SpecialFunc None
   Method _m_Alarms: Id {c0cf83f3-e704-4016-bd6f-2d30156087ff}
   Method _m_AutomaticControl: Id {ee0253ab-2fda-4db0-933c-ed048e84d0ed}
   Method _m_CmdCloseInnerDoor: Id {410bcb72-5351-4d55-ac55-5d0e27ce8155}
   Method _m_CmdDockTB: Id {8e382bf6-1d32-4474-a8a5-7c183a3c7036}
   Method _m_CmdOpenInnerDoor: Id {8be47e79-6c29-4713-b252-eb11a6bb46fb}
   Method _m_CmdUndockTB: Id {b328f671-5464-49bf-836c-f1f93f3d32af}
   Method _m_Devices: Id {b43c077f-3abc-4642-868d-7667cd19393f}
   Method _m_Hmi: Id {5090ba0a-8e2b-4ba6-88b3-b451c7c7863d}
   Method _m_Init: Id {f248bb7d-4543-4fa5-93e5-377095a1130a}
   Method _m_Inputs: Id {15e5d91e-088b-4383-82aa-ad9257b81a9b}
   Method _m_ManualControl: Id {cf85508a-2caa-42ea-a56c-5902a15aaf22}
   Method _m_Outputs: Id {748b7abf-6524-428b-ad1f-dd34bf2d901c}
   Method _m_Params: Id {78648659-4a86-4875-84af-aa8b2b68e067}
   Method _m_SeqStartup: Id {c8d2def1-61a3-43d6-a687-bb0d54548919}
   Method m_Main: Id {13829dfc-fc98-4f3a-8520-8dee66cb84d9}
   Method m_ReqCloseInnerDoor: Id {1fa4ee8a-afe9-445a-a083-5023c47af3e8}
   Method m_ReqDockTB: Id {a0624d17-910f-46f4-aad8-ec9dc796e335}
   Method m_ReqOpenInnerDoor: Id {af05bc54-8424-4586-adf6-51c519642be5}
   Method m_ReqUndockTB: Id {3ed99a4a-5538-4adf-806b-ec3280a600a5}
   Property p_bStaBoxAtDockedPosition: Id {95822bca-1047-492e-8877-1d8528242dc0}
   Get Get: Id {aa3a83b8-f468-44df-903c-150f557391f1}
   Property p_bStaBoxAtPreDockingPosition: Id {edbe1074-bded-474c-9558-f67f08872474}
   Get Get: Id {cf71d052-481e-48f0-aa51-5a234c033608}
   Property p_bStaDocked: Id {a61394df-c5f0-450a-8cdf-e47379cb8b81}
   Get Get: Id {e6843217-13bc-4765-b8f6-a237563e9d39}
   Property p_bStaDockingClampsClosed: Id {de32a338-e965-450c-a404-78adcd65d0d0}
   Get Get: Id {7682c14a-e4ab-4156-bdf2-ba42269377d9}
   Property p_bStaDockingClampsOpened: Id {20b689ca-7b07-4e51-a3ea-324f8cec92e0}
   Get Get: Id {31c09844-15c2-48d5-9a5b-8c43458c7d91}
   Property p_bStaDockingPositionFree: Id {1c1bcc1f-d42b-48d2-9743-d0c845e1b595}
   Get Get: Id {8f44ecfc-2d8a-4e22-a3b9-d3876337bbab}
   Property p_bStaInnerDoorClosedAndLocked: Id {dd31784c-49d6-4d32-a02f-66ee1e524851}
   Get Get: Id {ec81e0aa-07a2-4a59-858a-8a8d7988d797}
   Property p_bStaInnerDoorOpenedAndReleased: Id {38547cf9-5983-403c-914e-3b92e4e4e9d8}
   Get Get: Id {c2f8547d-c997-4c85-95f1-ef32b94df578}
   Property p_bStaUndocked: Id {2a632f80-434e-4ff6-ad02-3973770d7bbf}
   Get Get: Id {56b7d6e8-1510-46ea-84c2-20aa46607960} *)
